INTERFACE IEventHandler_OnAssertionFailed EXTENDS IEventHandlerBase

METHOD OnAssertionFailed
VAR_INPUT
    EventArgs   : IStreamReader;
END_VAR
END_METHOD

END_INTERFACE

(* stored: Version 1.1.0.1, ProductVersion 3.1.4024.3
   Itf IEventHandler_OnAssertionFailed: Id {1beeb754-b882-4909-9758-01ed67b6e663}
   Method OnAssertionFailed: Id {a43394cd-1082-4324-9c02-c866b6ff440c} *)
